# EPICS autosave request: iocBoot/iocUSBERB24/auto_settings.req
file "USBERB24_settings.req", P=$(P)
